FUNCTION_BLOCK Pid_Tests EXTENDS FB_TestSuite
VAR
    delta : LREAL := 1E-5;
END_VAR

OnlyProportionalPart();
OnlyPropotionalPartRunTwiceWithDifferentInputs();
OnlyIntegralPart();
OnlyIntegralPartSetPreviousIntegralPartBefore();
OnlyDifferentialPart();
OnlyDifferentialPartWithDiffLimit();
DifferentCycleTimesSameOutputIntegralPart();
DifferentCycleTimesSameOutputDifferentialPart();
DivideByZeroCycleTimeCheck();

METHOD DifferentCycleTimesSameOutputDifferentialPart
VAR_INST
    Pfast : PidController;
    Pslow : PidController;
    parameters : PidParameters := (Kd:=1);
    i : INT;
END_VAR
TEST('DifferentCycleTimesSameOutputDifferentialPart');

Pfast(parameters:=parameters, cycleTime:=1);
FOR i := 1 TO 4 DO
    Pfast.Update(setpoint:=3, actual:=2 + i * 0.25);
END_FOR

Pslow(parameters:=parameters, cycleTime:=2);
FOR i := 1 TO 2 DO
    Pslow.Update(setpoint:=3, actual:=2 + i * 0.5);
END_FOR

AssertEquals_LREAL(
    Expected:=Pslow.Out,
    Actual:=Pfast.Out,
    Delta:=delta,
    Message:='Slow and fast pid should give the same result'
);

TcUnit.TEST_FINISHED();
END_METHOD

METHOD DifferentCycleTimesSameOutputIntegralPart
VAR_INST
    Pfast : PidController;
    Pslow : PidController;
    parameters : PidParameters := (Ki:=1);
END_VAR
TEST('DifferentCycleTimesSameOutputIntegralPart');

Pfast(parameters:=parameters, cycleTime:=1);
Pfast.Update(setpoint:=3, actual:=2);
Pfast.Update(setpoint:=3, actual:=2);
Pslow(parameters:=parameters, cycleTime:=2);
Pslow.Update(setpoint:=3, actual:=2);

AssertEquals_LREAL(
    Expected:=Pslow.Out,
    Actual:=Pfast.Out,
    Delta:=delta,
    Message:='Slow and fast pid should give the same result'
);

TcUnit.TEST_FINISHED();
END_METHOD

METHOD DivideByZeroCycleTimeCheck
VAR_INST
    P : PidController;
END_VAR
TcUnit.TEST('DivideByZeroCycleTimeCheck');

P(cycleTime:=0);
P.Update(setpoint:=1, actual:=1);

//Should not cause an exception

TcUnit.TEST_FINISHED();
END_METHOD

METHOD OnlyDifferentialPart
VAR_INST
    P : PidController;
    parameters : PidParameters := (Kd:=0.01);
END_VAR
TcUnit.TEST('OnlyDifferentialPart');

P(parameters:=parameters);
P.Update(setpoint:=10, actual:=6);
AssertEquals_LREAL(
    Expected:=0.04,
    Actual:=P.Out,
    Delta:=delta,
    Message:='Pid output run 1 not correct'
);

P.Update(setpoint:=10, actual:=8);
AssertEquals_LREAL(
    Expected:=-0.02,
    Actual:=P.Out,
    Delta:=delta,
    Message:='Pid output run 2 not correct'
);

TcUnit.TEST_FINISHED();
END_METHOD

METHOD OnlyDifferentialPartWithDiffLimit
VAR_INST
    P : PidController;
    parameters : PidParameters := (Kd:=0.01);
END_VAR
TcUnit.TEST('OnlyDifferentialPartWithDiffLimit');

P.DifferentialPartLimit := 3;
P(parameters:=parameters);
P.Update(setpoint:=10, actual:=6);
AssertEquals_LREAL(
    Expected:=0,
    Actual:=P.Out,
    Delta:=delta,
    Message:='Pid output run 1 not correct'
);

P.Update(setpoint:=10, actual:=8);
AssertEquals_LREAL(
    Expected:=-0.02,
    Actual:=P.Out,
    Delta:=delta,
    Message:='Pid output run 2 not correct'
);

TcUnit.TEST_FINISHED();
END_METHOD

METHOD OnlyIntegralPart
VAR_INST
    P : PidController := (cycleTime:=1);
    parameters : PidParameters := (Ki:=0.25);
END_VAR
TcUnit.TEST('OnlyIntegralPart');

P(parameters:=parameters);
P.Update(setpoint:=10, actual:=6);
AssertEquals_LREAL(
    Expected:=1,
    Actual:=P.Out,
    Delta:=delta,
    Message:='Pid output run 1 not correct'
);

P.Update(setpoint:=10, actual:=8);
AssertEquals_LREAL(
    Expected:=1.5,
    Actual:=P.Out,
    Delta:=delta,
    Message:='Pid output run 2 not correct'
);

TcUnit.TEST_FINISHED();
END_METHOD

METHOD OnlyIntegralPartSetPreviousIntegralPartBefore
VAR_INST
    P : PidController := (cycleTime:=1);
    parameters : PidParameters := (Ki:=0.25);
END_VAR
TcUnit.TEST('OnlyIntegralPartSetPreviousIntegralPartBefore');

P.PreviousIntegralPart := 3;
P(parameters:=parameters);
P.Update(setpoint:=10, actual:=6);
AssertEquals_LREAL(
    Expected:=4,
    Actual:=P.Out,
    Delta:=delta,
    Message:='Pid output run 1 not correct'
);

P.Update(setpoint:=10, actual:=8);
AssertEquals_LREAL(
    Expected:=4.5,
    Actual:=P.Out,
    Delta:=delta,
    Message:='Pid output run 2 not correct'
);

TcUnit.TEST_FINISHED();
END_METHOD

METHOD OnlyProportionalPart
VAR_INST
    P : PidController;
    parameters : PidParameters := (Kp:=5);
END_VAR
TcUnit.TEST('OnlyProportionalPart');

P(parameters:=parameters);
P.Update(setpoint:=10, actual:=5);

AssertEquals_LREAL(Expected:=25, Actual:=P.Out, Delta:=delta, Message:='Pid output not correct');

TcUnit.TEST_FINISHED();
END_METHOD

METHOD OnlyPropotionalPartRunTwiceWithDifferentInputs
VAR_INST
    P : PidController;
    parameters : PidParameters := (Kp:=2);
END_VAR
TcUnit.TEST('OnlyPropotionalPartRunTwiceWithDifferentInputs');

P(parameters:=parameters);
P.Update(setpoint:=3, actual:=4.5);

AssertEquals_LREAL(
    Expected:=-3,
    Actual:=P.Out,
    Delta:=delta,
    Message:='Pid output after run 1 not correct'
);

P.Update(setpoint:=-8, actual:=-6);

AssertEquals_LREAL(
    Expected:=-4,
    Actual:=P.Out,
    Delta:=delta,
    Message:='Pid output after run 2 not correct'
);

TcUnit.TEST_FINISHED();
END_METHOD

END_FUNCTION_BLOCK

(* stored: Version 1.1.0.1, ProductVersion 3.1.4024.12
   POU Pid_Tests: Id {d37e3a2d-290f-492c-9ef6-af8dd98f69e3}, SpecialFunc None
   Method DifferentCycleTimesSameOutputDifferentialPart: Id {21fb58cc-afc4-4d4c-bfea-12ac57e21910}
   Method DifferentCycleTimesSameOutputIntegralPart: Id {07c9ad63-6800-4d52-804c-298e0cae3bb9}
   Method DivideByZeroCycleTimeCheck: Id {cc32b3cb-eb63-4350-bd0f-4654057ba87c}
   Method OnlyDifferentialPart: Id {4f99075d-a13f-4f18-8a15-c8ddba8e5a52}
   Method OnlyDifferentialPartWithDiffLimit: Id {241d286d-fea2-4eb4-8a87-6d9bdc37a17d}
   Method OnlyIntegralPart: Id {5d97b5ea-7ca7-495f-b7ce-68e585bdb9a4}
   Method OnlyIntegralPartSetPreviousIntegralPartBefore: Id {e14023e9-bbe5-4ab4-b516-86db5b89a50c}
   Method OnlyProportionalPart: Id {4180392b-050f-4fed-a265-d9a44e45b893}
   Method OnlyPropotionalPartRunTwiceWithDifferentInputs: Id {1d265881-ea1f-4b87-98ee-c292edfec96c} *)
